// TIA Portal V17 export
// export: Created 2024-09-02T12:50:24.6153138Z, ExportSetting WithDefaults, DisplayName Totally Integrated Automation Portal, DisplayVersion V17, DisplayName TIA Portal Openness, DisplayVersion V17, DisplayName TIA Portal Version Control Interface, DisplayVersion V17, DisplayName STEP 7 Professional, DisplayVersion V17, DisplayName STEP 7 Safety, DisplayVersion V17, DisplayName WinCC Professional, DisplayVersion V17
FUNCTION "Energy_And_Air_Counter" : Void   // FC23, LAD
{ S7_Optimized_Access := 'TRUE' }
VERSION : 0.1
// stored: AutoNumber false, IsIECCheckEnabled false, SetENOAutomatically false, UDAEnableTagReadback false
   VAR_INPUT
      Active_Air : DInt;
      Active_Energy : LReal;
      Reset_total : Bool;
      Reset_Time_Stamp : Bool;
      Count_Part : Bool;
   END_VAR
   VAR_TEMP
      Active_En_KWh : LReal;
      Active_En_M3 : Real;
      tActive_En_M3 : Real;
      Reset_periods_Energy : Bool;
      Number : Int;
      temp : Int;
      t_Move_data : Bool;
      tReset_total : Bool;
   END_VAR
   VAR_TEMP   // added for the SCL form of the ladder/FBD networks
      _w1 : Bool;
      _w2 : Bool;
      _w3 : Bool;
   END_VAR
BEGIN

REGION Network 1: Actual_Active_Energy
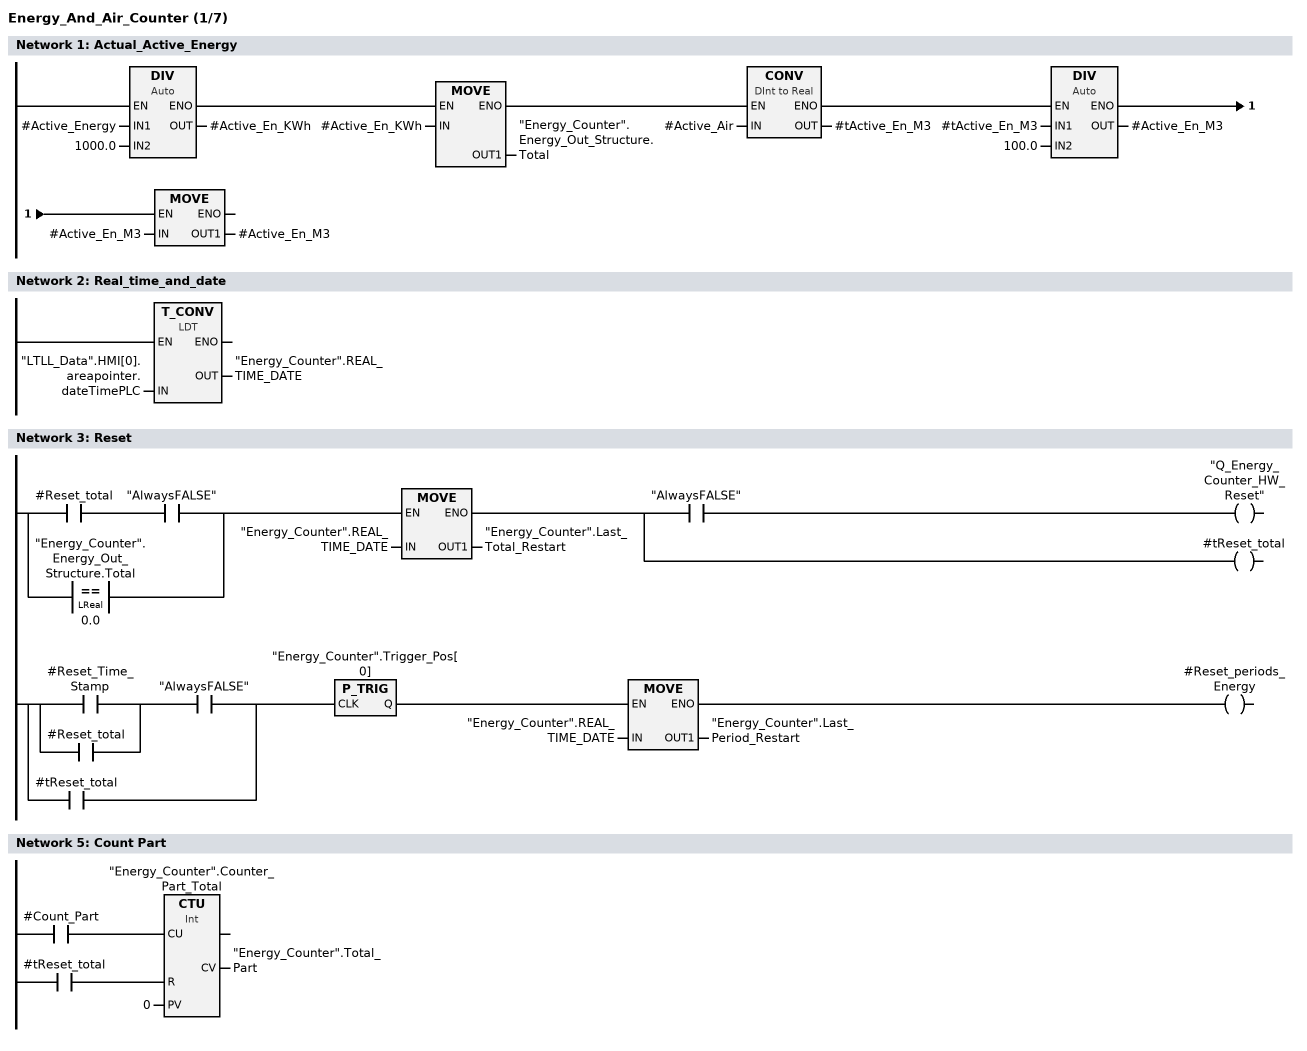
   RUNG wire#powerrail
      Div(in1 := #Active_Energy, in2 := 1000.0, out => #Active_En_KWh)
      Move(in := #Active_En_KWh, out1 => "Energy_Counter".Energy_Out_Structure.Total)
      { S7_Templates := "[SrcType := DInt, DestType := Real]" } Convert(in := #Active_Air, out => #tActive_En_M3)
      Div(in1 := #tActive_En_M3, in2 := 100.0, out => #Active_En_M3)
      Move(in := #Active_En_M3, out1 => #Active_En_M3)
   END_RUNG
   // the same network as SCL:
   #Active_En_KWh := #Active_Energy / 1000.0;
   "Energy_Counter".Energy_Out_Structure.Total := #Active_En_KWh;
   #tActive_En_M3 := DINT_TO_REAL(#Active_Air);
   #Active_En_M3 := #tActive_En_M3 / 100.0;
   #Active_En_M3 := #Active_En_M3;
END_REGION

REGION Network 2: Real_time_and_date
   RUNG wire#powerrail
      { S7_Templates := "[src_type := LDT, dest_type := DTL]" } T_CONV(IN := "LTLL_Data".HMI[0].areapointer.dateTimePLC, OUT => "Energy_Counter".REAL_TIME_DATE)
   END_RUNG
   // the same network as SCL:
   T_CONV(IN := "LTLL_Data".HMI[0].areapointer.dateTimePLC, OUT => "Energy_Counter".REAL_TIME_DATE);
END_REGION

REGION Network 3: Reset
   RUNG wire#powerrail
      Contact( #Reset_total )
      Contact( "AlwaysFALSE" )
      wire#w1
      Move(in := "Energy_Counter".REAL_TIME_DATE, out1 => "Energy_Counter".Last_Total_Restart)
      wire#w2
      Contact( "AlwaysFALSE" )
      Coil( "Q_Energy_Counter_HW_Reset" )
   END_RUNG
   RUNG wire#powerrail
      { S7_Templates := "SrcType := LReal" } EQ_Contact(in1 := "Energy_Counter".Energy_Out_Structure.Total, in2 := 0.0)
   END_RUNG wire#w1
   RUNG wire#w2
      Coil( #tReset_total )
   END_RUNG
   RUNG wire#powerrail
      Contact( #Reset_Time_Stamp )
      wire#w3
      Contact( "AlwaysFALSE" )
      wire#w4
      P_Trig( "Energy_Counter".Trigger_Pos[0] )
      Move(in := "Energy_Counter".REAL_TIME_DATE, out1 => "Energy_Counter".Last_Period_Restart)
      Coil( #Reset_periods_Energy )
   END_RUNG
   RUNG wire#powerrail
      Contact( #Reset_total )
   END_RUNG wire#w3
   RUNG wire#powerrail
      Contact( #tReset_total )
   END_RUNG wire#w4
   // the same network as SCL:
   #_w1 := (#Reset_total AND "AlwaysFALSE") OR ("Energy_Counter".Energy_Out_Structure.Total = 0.0);
   IF #_w1 THEN "Energy_Counter".Last_Total_Restart := "Energy_Counter".REAL_TIME_DATE; END_IF;
   "Q_Energy_Counter_HW_Reset" := #_w1 AND "AlwaysFALSE";
   #tReset_total := #_w1;
   #_w2 := ((#Reset_Time_Stamp OR #Reset_total) AND "AlwaysFALSE") OR #tReset_total;
   #_w3 := #_w2 AND NOT "Energy_Counter".Trigger_Pos[0];   // rising edge
   "Energy_Counter".Trigger_Pos[0] := #_w2;
   IF #_w3 THEN "Energy_Counter".Last_Period_Restart := "Energy_Counter".REAL_TIME_DATE; END_IF;
   #Reset_periods_Energy := #_w3;
END_REGION

REGION Network 4: ########### Part Counting #########
END_REGION

REGION Network 5: Count Part
   RUNG wire#powerrail
      Contact( #Count_Part )
      { S7_Templates := "value_type := Int" } "Energy_Counter".Counter_Part_Total.CTU(r := wire#w1, pv := 0, cv => "Energy_Counter".Total_Part)
   END_RUNG
   RUNG wire#powerrail
      Contact( #tReset_total )
   END_RUNG wire#w1
   // the same network as SCL:
   "Energy_Counter".Counter_Part_Total.CTU(CU := #Count_Part,
                           R := #tReset_total,
                           PV := 0,
                           CV => "Energy_Counter".Total_Part);
END_REGION

REGION Network 6: Total Energi / Air per Part
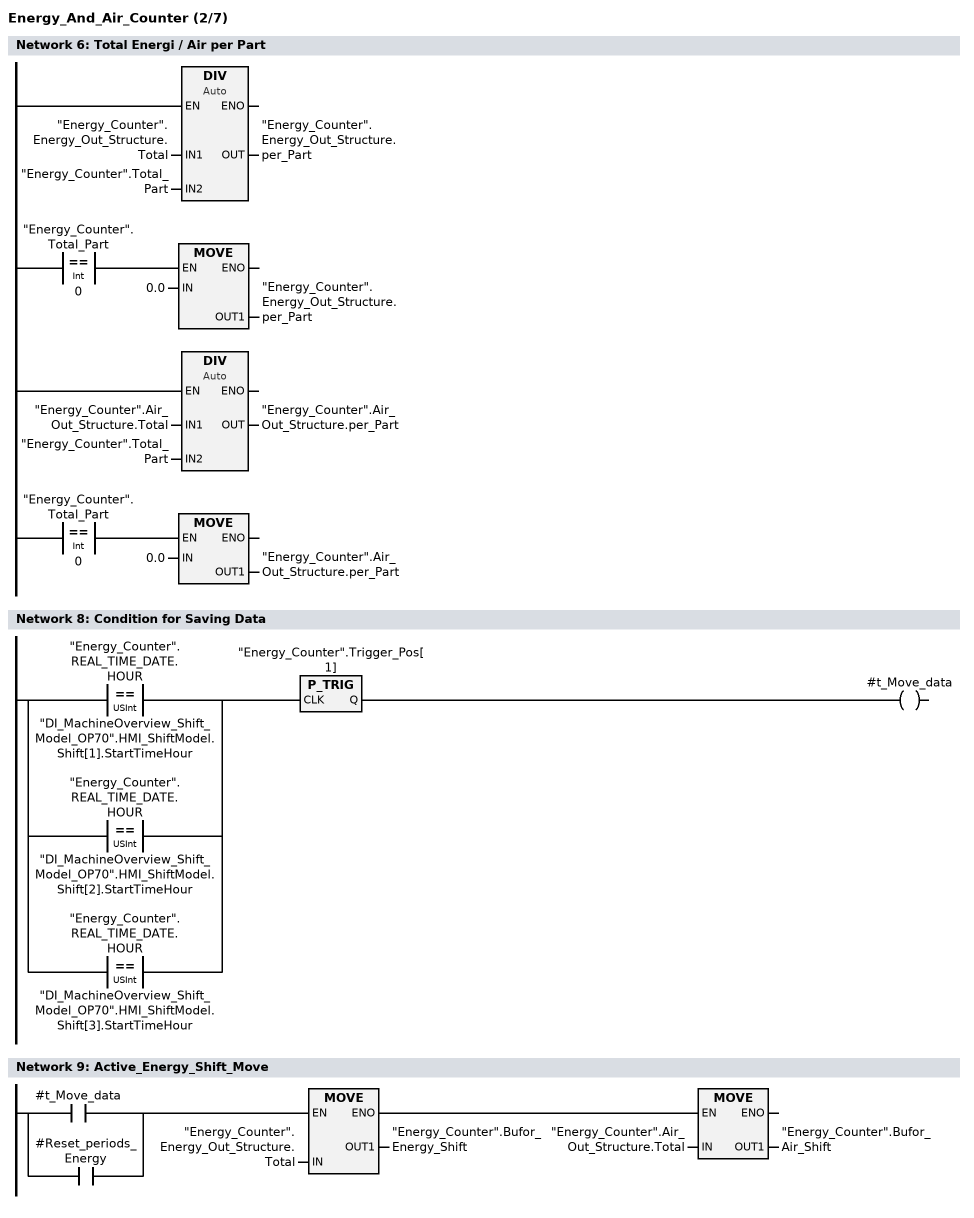
   RUNG wire#powerrail
      Div(in1 := "Energy_Counter".Energy_Out_Structure.Total, in2 := "Energy_Counter".Total_Part, out => "Energy_Counter".Energy_Out_Structure.per_Part)
   END_RUNG
   RUNG wire#powerrail
      { S7_Templates := "SrcType := Int" } EQ_Contact(in1 := "Energy_Counter".Total_Part, in2 := 0)
      Move(in := 0.0, out1 => "Energy_Counter".Energy_Out_Structure.per_Part)
   END_RUNG
   RUNG wire#powerrail
      Div(in1 := "Energy_Counter".Air_Out_Structure.Total, in2 := "Energy_Counter".Total_Part, out => "Energy_Counter".Air_Out_Structure.per_Part)
   END_RUNG
   RUNG wire#powerrail
      { S7_Templates := "SrcType := Int" } EQ_Contact(in1 := "Energy_Counter".Total_Part, in2 := 0)
      Move(in := 0.0, out1 => "Energy_Counter".Air_Out_Structure.per_Part)
   END_RUNG
   // the same network as SCL:
   "Energy_Counter".Energy_Out_Structure.per_Part := "Energy_Counter".Energy_Out_Structure.Total / "Energy_Counter".Total_Part;
   IF "Energy_Counter".Total_Part = 0 THEN "Energy_Counter".Energy_Out_Structure.per_Part := 0.0; END_IF;
   "Energy_Counter".Air_Out_Structure.per_Part := "Energy_Counter".Air_Out_Structure.Total / "Energy_Counter".Total_Part;
   IF "Energy_Counter".Total_Part = 0 THEN "Energy_Counter".Air_Out_Structure.per_Part := 0.0; END_IF;
END_REGION

REGION Network 7: ########### ENERGY PER SHIFT #########
END_REGION

REGION Network 8: Condition for Saving Data
   RUNG wire#powerrail
      { S7_Templates := "SrcType := USInt" } EQ_Contact(in1 := "Energy_Counter".REAL_TIME_DATE.HOUR, in2 := "DI_MachineOverview_Shift_Model_OP70".HMI_ShiftModel.Shift[1].StartTimeHour)
      wire#w1
      P_Trig( "Energy_Counter".Trigger_Pos[1] )
      Coil( #t_Move_data )
   END_RUNG
   RUNG wire#powerrail
      { S7_Templates := "SrcType := USInt" } EQ_Contact(in1 := "Energy_Counter".REAL_TIME_DATE.HOUR, in2 := "DI_MachineOverview_Shift_Model_OP70".HMI_ShiftModel.Shift[2].StartTimeHour)
   END_RUNG wire#w1
   RUNG wire#powerrail
      { S7_Templates := "SrcType := USInt" } EQ_Contact(in1 := "Energy_Counter".REAL_TIME_DATE.HOUR, in2 := "DI_MachineOverview_Shift_Model_OP70".HMI_ShiftModel.Shift[3].StartTimeHour)
   END_RUNG wire#w1
   // the same network as SCL:
   #_w1 := ("Energy_Counter".REAL_TIME_DATE.HOUR = "DI_MachineOverview_Shift_Model_OP70".HMI_ShiftModel.Shift[1].StartTimeHour) OR ("Energy_Counter".REAL_TIME_DATE.HOUR = "DI_MachineOverview_Shift_Model_OP70".HMI_ShiftModel.Shift[2].StartTimeHour) OR ("Energy_Counter".REAL_TIME_DATE.HOUR = "DI_MachineOverview_Shift_Model_OP70".HMI_ShiftModel.Shift[3].StartTimeHour);
   #_w2 := #_w1 AND NOT "Energy_Counter".Trigger_Pos[1];   // rising edge
   "Energy_Counter".Trigger_Pos[1] := #_w1;
   #t_Move_data := #_w2;
END_REGION

REGION Network 9: Active_Energy_Shift_Move
   RUNG wire#powerrail
      Contact( #t_Move_data )
      wire#w1
      Move(in := "Energy_Counter".Energy_Out_Structure.Total, out1 => "Energy_Counter".Bufor_Energy_Shift)
      Move(in := "Energy_Counter".Air_Out_Structure.Total, out1 => "Energy_Counter".Bufor_Air_Shift)
   END_RUNG
   RUNG wire#powerrail
      Contact( #Reset_periods_Energy )
   END_RUNG wire#w1
   // the same network as SCL:
   IF #t_Move_data OR #Reset_periods_Energy THEN
       "Energy_Counter".Bufor_Energy_Shift := "Energy_Counter".Energy_Out_Structure.Total;
       "Energy_Counter".Bufor_Air_Shift := "Energy_Counter".Air_Out_Structure.Total;
   END_IF;
END_REGION

REGION Network 10: Calculation
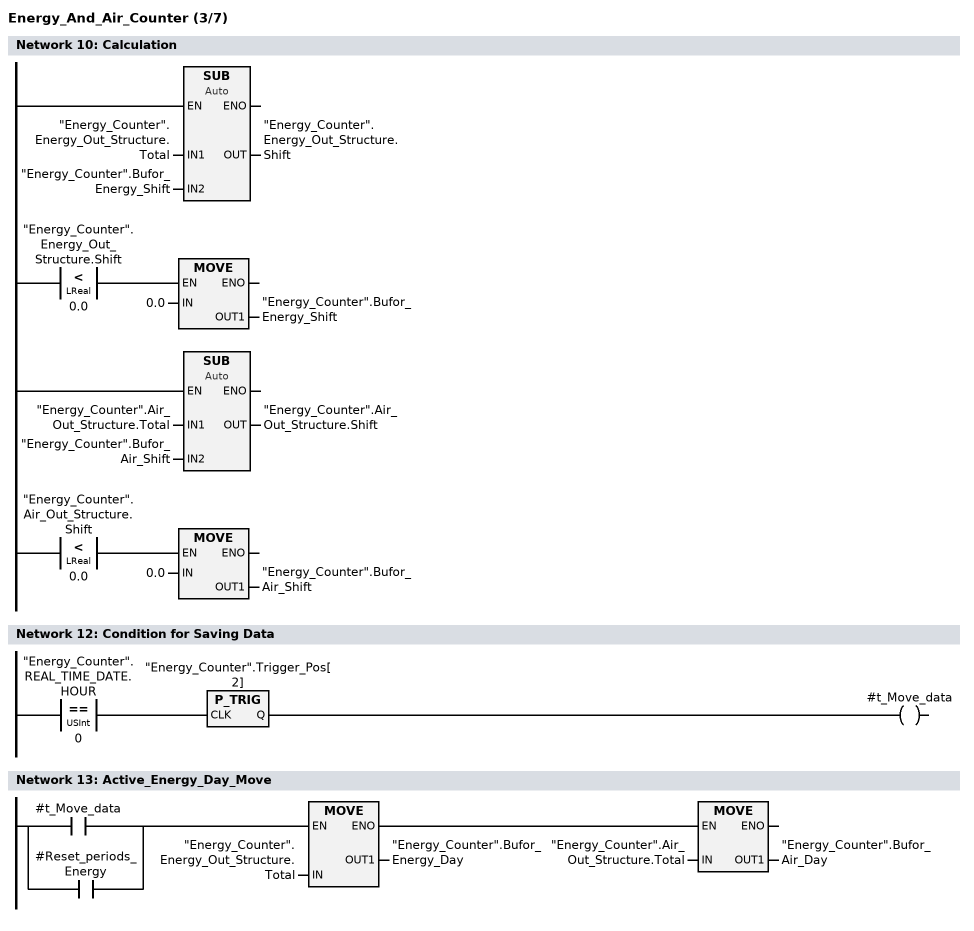
   RUNG wire#powerrail
      Sub(in1 := "Energy_Counter".Energy_Out_Structure.Total, in2 := "Energy_Counter".Bufor_Energy_Shift, out => "Energy_Counter".Energy_Out_Structure.Shift)
   END_RUNG
   RUNG wire#powerrail
      { S7_Templates := "SrcType := LReal" } LT_Contact(in1 := "Energy_Counter".Energy_Out_Structure.Shift, in2 := 0.0)
      Move(in := 0.0, out1 => "Energy_Counter".Bufor_Energy_Shift)
   END_RUNG
   RUNG wire#powerrail
      Sub(in1 := "Energy_Counter".Air_Out_Structure.Total, in2 := "Energy_Counter".Bufor_Air_Shift, out => "Energy_Counter".Air_Out_Structure.Shift)
   END_RUNG
   RUNG wire#powerrail
      { S7_Templates := "SrcType := LReal" } LT_Contact(in1 := "Energy_Counter".Air_Out_Structure.Shift, in2 := 0.0)
      Move(in := 0.0, out1 => "Energy_Counter".Bufor_Air_Shift)
   END_RUNG
   // the same network as SCL:
   "Energy_Counter".Energy_Out_Structure.Shift := "Energy_Counter".Energy_Out_Structure.Total - "Energy_Counter".Bufor_Energy_Shift;
   IF "Energy_Counter".Energy_Out_Structure.Shift < 0.0 THEN
       "Energy_Counter".Bufor_Energy_Shift := 0.0;
   END_IF;
   "Energy_Counter".Air_Out_Structure.Shift := "Energy_Counter".Air_Out_Structure.Total - "Energy_Counter".Bufor_Air_Shift;
   IF "Energy_Counter".Air_Out_Structure.Shift < 0.0 THEN "Energy_Counter".Bufor_Air_Shift := 0.0; END_IF;
END_REGION

REGION Network 11: ########### ENERGY PER DAY #########
END_REGION

REGION Network 12: Condition for Saving Data
   RUNG wire#powerrail
      { S7_Templates := "SrcType := USInt" } EQ_Contact(in1 := "Energy_Counter".REAL_TIME_DATE.HOUR, in2 := 0)
      P_Trig( "Energy_Counter".Trigger_Pos[2] )
      Coil( #t_Move_data )
   END_RUNG
   // the same network as SCL:
   #_w1 := "Energy_Counter".REAL_TIME_DATE.HOUR = 0;
   #_w2 := #_w1 AND NOT "Energy_Counter".Trigger_Pos[2];   // rising edge
   "Energy_Counter".Trigger_Pos[2] := #_w1;
   #t_Move_data := #_w2;
END_REGION

REGION Network 13: Active_Energy_Day_Move
   RUNG wire#powerrail
      Contact( #t_Move_data )
      wire#w1
      Move(in := "Energy_Counter".Energy_Out_Structure.Total, out1 => "Energy_Counter".Bufor_Energy_Day)
      Move(in := "Energy_Counter".Air_Out_Structure.Total, out1 => "Energy_Counter".Bufor_Air_Day)
   END_RUNG
   RUNG wire#powerrail
      Contact( #Reset_periods_Energy )
   END_RUNG wire#w1
   // the same network as SCL:
   IF #t_Move_data OR #Reset_periods_Energy THEN
       "Energy_Counter".Bufor_Energy_Day := "Energy_Counter".Energy_Out_Structure.Total;
       "Energy_Counter".Bufor_Air_Day := "Energy_Counter".Air_Out_Structure.Total;
   END_IF;
END_REGION

REGION Network 14: Calculation
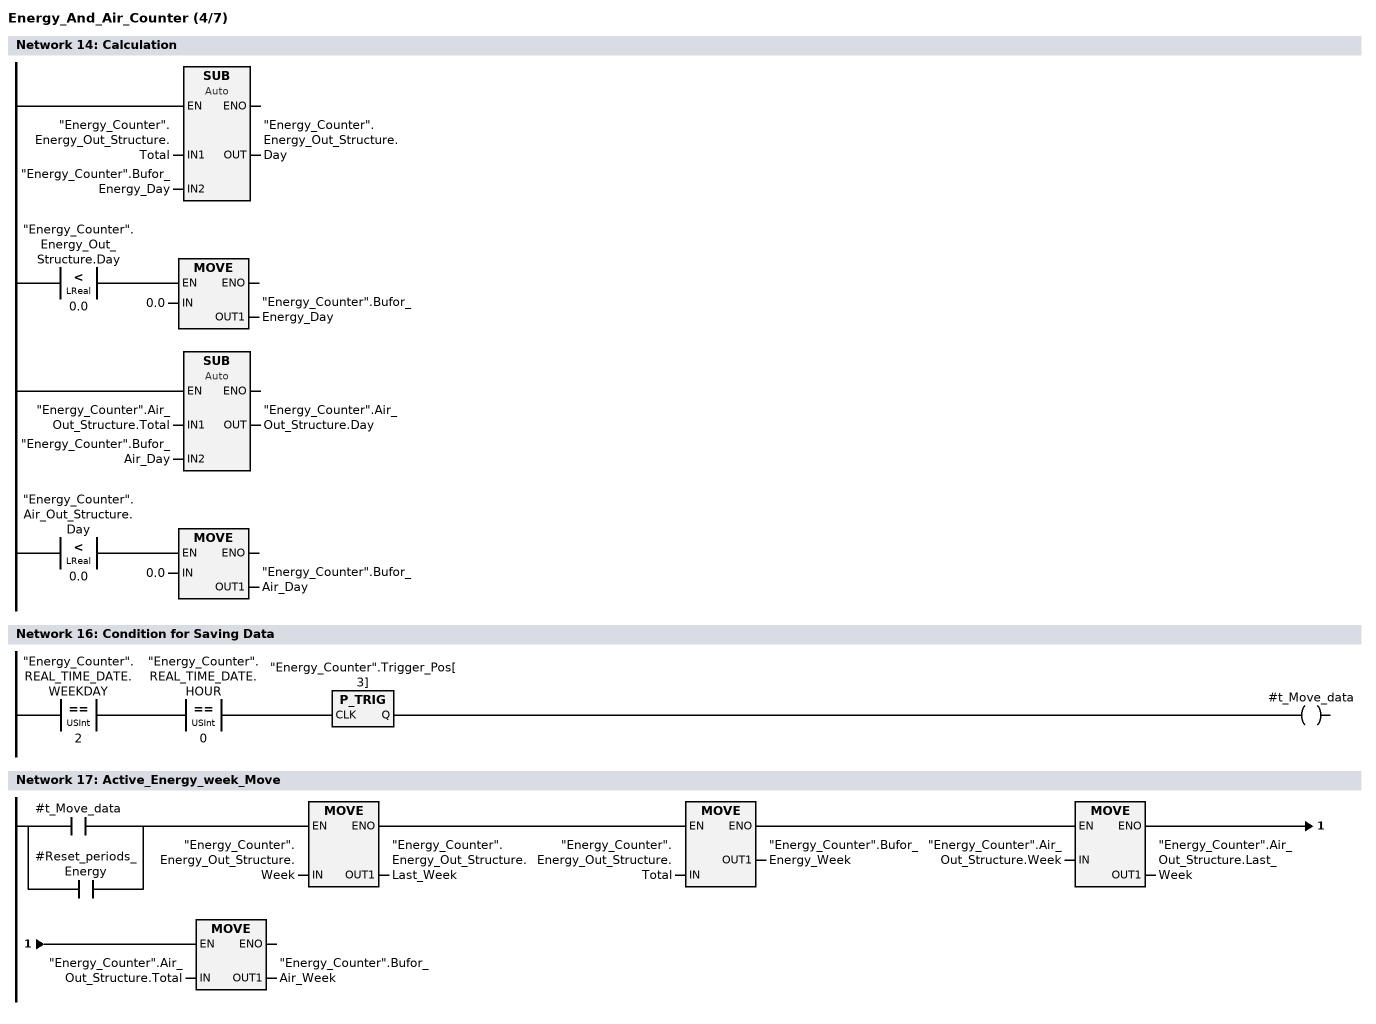
   RUNG wire#powerrail
      Sub(in1 := "Energy_Counter".Energy_Out_Structure.Total, in2 := "Energy_Counter".Bufor_Energy_Day, out => "Energy_Counter".Energy_Out_Structure.Day)
   END_RUNG
   RUNG wire#powerrail
      { S7_Templates := "SrcType := LReal" } LT_Contact(in1 := "Energy_Counter".Energy_Out_Structure.Day, in2 := 0.0)
      Move(in := 0.0, out1 => "Energy_Counter".Bufor_Energy_Day)
   END_RUNG
   RUNG wire#powerrail
      Sub(in1 := "Energy_Counter".Air_Out_Structure.Total, in2 := "Energy_Counter".Bufor_Air_Day, out => "Energy_Counter".Air_Out_Structure.Day)
   END_RUNG
   RUNG wire#powerrail
      { S7_Templates := "SrcType := LReal" } LT_Contact(in1 := "Energy_Counter".Air_Out_Structure.Day, in2 := 0.0)
      Move(in := 0.0, out1 => "Energy_Counter".Bufor_Air_Day)
   END_RUNG
   // the same network as SCL:
   "Energy_Counter".Energy_Out_Structure.Day := "Energy_Counter".Energy_Out_Structure.Total - "Energy_Counter".Bufor_Energy_Day;
   IF "Energy_Counter".Energy_Out_Structure.Day < 0.0 THEN "Energy_Counter".Bufor_Energy_Day := 0.0; END_IF;
   "Energy_Counter".Air_Out_Structure.Day := "Energy_Counter".Air_Out_Structure.Total - "Energy_Counter".Bufor_Air_Day;
   IF "Energy_Counter".Air_Out_Structure.Day < 0.0 THEN "Energy_Counter".Bufor_Air_Day := 0.0; END_IF;
END_REGION

REGION Network 15: ########### ENERGY PER WEEK #########
END_REGION

REGION Network 16: Condition for Saving Data
   RUNG wire#powerrail
      { S7_Templates := "SrcType := USInt" } EQ_Contact(in1 := "Energy_Counter".REAL_TIME_DATE.WEEKDAY, in2 := 2)
      { S7_Templates := "SrcType := USInt" } EQ_Contact(in1 := "Energy_Counter".REAL_TIME_DATE.HOUR, in2 := 0)
      P_Trig( "Energy_Counter".Trigger_Pos[3] )
      Coil( #t_Move_data )
   END_RUNG
   // the same network as SCL:
   #_w1 := ("Energy_Counter".REAL_TIME_DATE.WEEKDAY = 2) AND ("Energy_Counter".REAL_TIME_DATE.HOUR = 0);
   #_w2 := #_w1 AND NOT "Energy_Counter".Trigger_Pos[3];   // rising edge
   "Energy_Counter".Trigger_Pos[3] := #_w1;
   #t_Move_data := #_w2;
END_REGION

REGION Network 17: Active_Energy_week_Move
   RUNG wire#powerrail
      Contact( #t_Move_data )
      wire#w1
      Move(in := "Energy_Counter".Energy_Out_Structure.Week, out1 => "Energy_Counter".Energy_Out_Structure.Last_Week)
      Move(in := "Energy_Counter".Energy_Out_Structure.Total, out1 => "Energy_Counter".Bufor_Energy_Week)
      Move(in := "Energy_Counter".Air_Out_Structure.Week, out1 => "Energy_Counter".Air_Out_Structure.Last_Week)
      Move(in := "Energy_Counter".Air_Out_Structure.Total, out1 => "Energy_Counter".Bufor_Air_Week)
   END_RUNG
   RUNG wire#powerrail
      Contact( #Reset_periods_Energy )
   END_RUNG wire#w1
   // the same network as SCL:
   IF #t_Move_data OR #Reset_periods_Energy THEN
       "Energy_Counter".Energy_Out_Structure.Last_Week := "Energy_Counter".Energy_Out_Structure.Week;
       "Energy_Counter".Bufor_Energy_Week := "Energy_Counter".Energy_Out_Structure.Total;
       "Energy_Counter".Air_Out_Structure.Last_Week := "Energy_Counter".Air_Out_Structure.Week;
       "Energy_Counter".Bufor_Air_Week := "Energy_Counter".Air_Out_Structure.Total;
   END_IF;
END_REGION

REGION Network 18: Calculation
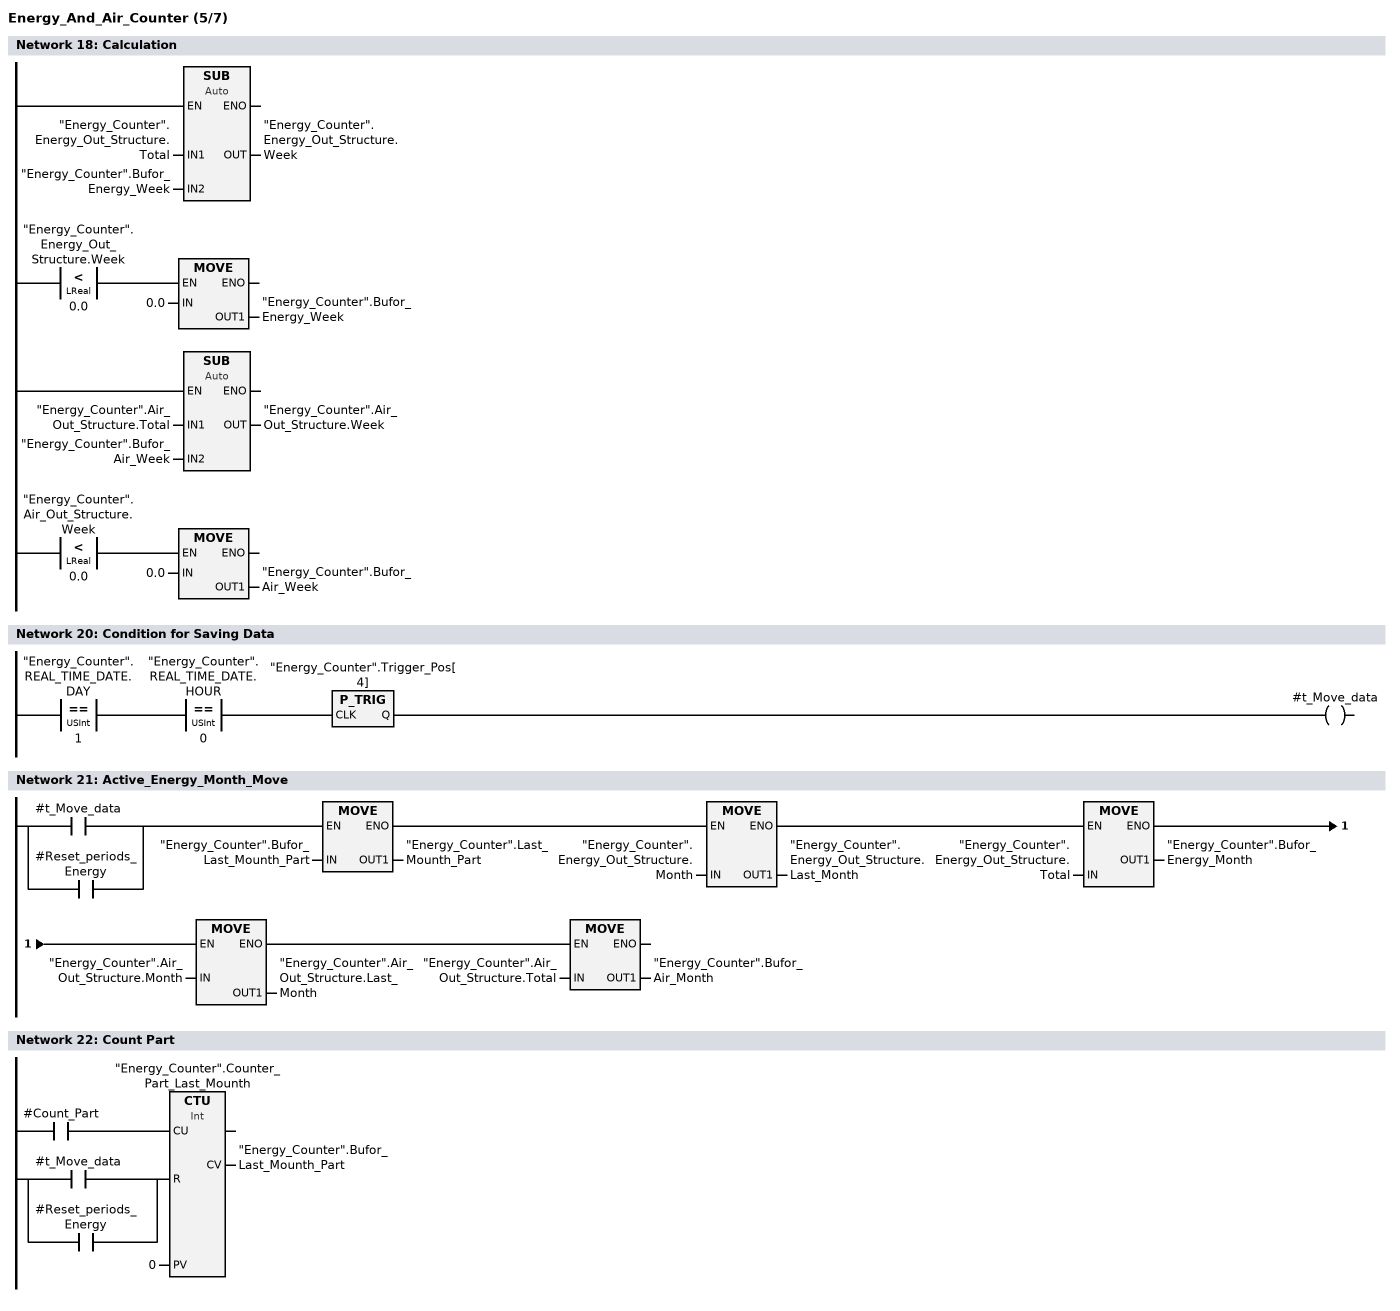
   RUNG wire#powerrail
      Sub(in1 := "Energy_Counter".Energy_Out_Structure.Total, in2 := "Energy_Counter".Bufor_Energy_Week, out => "Energy_Counter".Energy_Out_Structure.Week)
   END_RUNG
   RUNG wire#powerrail
      { S7_Templates := "SrcType := LReal" } LT_Contact(in1 := "Energy_Counter".Energy_Out_Structure.Week, in2 := 0.0)
      Move(in := 0.0, out1 => "Energy_Counter".Bufor_Energy_Week)
   END_RUNG
   RUNG wire#powerrail
      Sub(in1 := "Energy_Counter".Air_Out_Structure.Total, in2 := "Energy_Counter".Bufor_Air_Week, out => "Energy_Counter".Air_Out_Structure.Week)
   END_RUNG
   RUNG wire#powerrail
      { S7_Templates := "SrcType := LReal" } LT_Contact(in1 := "Energy_Counter".Air_Out_Structure.Week, in2 := 0.0)
      Move(in := 0.0, out1 => "Energy_Counter".Bufor_Air_Week)
   END_RUNG
   // the same network as SCL:
   "Energy_Counter".Energy_Out_Structure.Week := "Energy_Counter".Energy_Out_Structure.Total - "Energy_Counter".Bufor_Energy_Week;
   IF "Energy_Counter".Energy_Out_Structure.Week < 0.0 THEN
       "Energy_Counter".Bufor_Energy_Week := 0.0;
   END_IF;
   "Energy_Counter".Air_Out_Structure.Week := "Energy_Counter".Air_Out_Structure.Total - "Energy_Counter".Bufor_Air_Week;
   IF "Energy_Counter".Air_Out_Structure.Week < 0.0 THEN "Energy_Counter".Bufor_Air_Week := 0.0; END_IF;
END_REGION

REGION Network 19: ########### ENERGY PER MONTH #########
END_REGION

REGION Network 20: Condition for Saving Data
   RUNG wire#powerrail
      { S7_Templates := "SrcType := USInt" } EQ_Contact(in1 := "Energy_Counter".REAL_TIME_DATE.DAY, in2 := 1)
      { S7_Templates := "SrcType := USInt" } EQ_Contact(in1 := "Energy_Counter".REAL_TIME_DATE.HOUR, in2 := 0)
      P_Trig( "Energy_Counter".Trigger_Pos[4] )
      Coil( #t_Move_data )
   END_RUNG
   // the same network as SCL:
   #_w1 := ("Energy_Counter".REAL_TIME_DATE.DAY = 1) AND ("Energy_Counter".REAL_TIME_DATE.HOUR = 0);
   #_w2 := #_w1 AND NOT "Energy_Counter".Trigger_Pos[4];   // rising edge
   "Energy_Counter".Trigger_Pos[4] := #_w1;
   #t_Move_data := #_w2;
END_REGION

REGION Network 21: Active_Energy_Month_Move
   RUNG wire#powerrail
      Contact( #t_Move_data )
      wire#w1
      Move(in := "Energy_Counter".Bufor_Last_Mounth_Part, out1 => "Energy_Counter".Last_Mounth_Part)
      Move(in := "Energy_Counter".Energy_Out_Structure.Month, out1 => "Energy_Counter".Energy_Out_Structure.Last_Month)
      Move(in := "Energy_Counter".Energy_Out_Structure.Total, out1 => "Energy_Counter".Bufor_Energy_Month)
      Move(in := "Energy_Counter".Air_Out_Structure.Month, out1 => "Energy_Counter".Air_Out_Structure.Last_Month)
      Move(in := "Energy_Counter".Air_Out_Structure.Total, out1 => "Energy_Counter".Bufor_Air_Month)
   END_RUNG
   RUNG wire#powerrail
      Contact( #Reset_periods_Energy )
   END_RUNG wire#w1
   // the same network as SCL:
   IF #t_Move_data OR #Reset_periods_Energy THEN
       "Energy_Counter".Last_Mounth_Part := "Energy_Counter".Bufor_Last_Mounth_Part;
       "Energy_Counter".Energy_Out_Structure.Last_Month := "Energy_Counter".Energy_Out_Structure.Month;
       "Energy_Counter".Bufor_Energy_Month := "Energy_Counter".Energy_Out_Structure.Total;
       "Energy_Counter".Air_Out_Structure.Last_Month := "Energy_Counter".Air_Out_Structure.Month;
       "Energy_Counter".Bufor_Air_Month := "Energy_Counter".Air_Out_Structure.Total;
   END_IF;
END_REGION

REGION Network 22: Count Part
   RUNG wire#powerrail
      Contact( #Count_Part )
      { S7_Templates := "value_type := Int" } "Energy_Counter".Counter_Part_Last_Mounth.CTU(r := wire#w1, pv := 0, cv => "Energy_Counter".Bufor_Last_Mounth_Part)
   END_RUNG
   RUNG wire#powerrail
      Contact( #t_Move_data )
   END_RUNG wire#w1
   RUNG wire#powerrail
      Contact( #Reset_periods_Energy )
   END_RUNG wire#w1
   // the same network as SCL:
   "Energy_Counter".Counter_Part_Last_Mounth.CTU(CU := #Count_Part,
                           R := #t_Move_data OR #Reset_periods_Energy,
                           PV := 0,
                           CV => "Energy_Counter".Bufor_Last_Mounth_Part);
END_REGION

REGION Network 23: Calculation
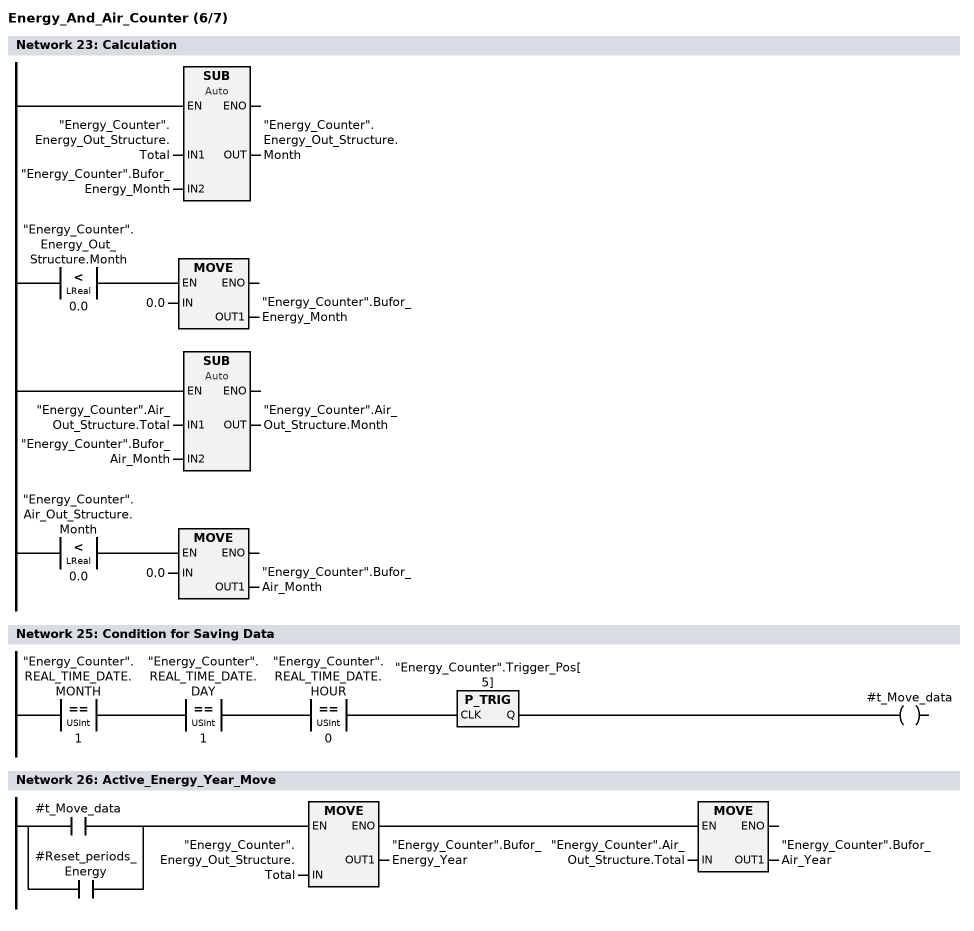
   RUNG wire#powerrail
      Sub(in1 := "Energy_Counter".Energy_Out_Structure.Total, in2 := "Energy_Counter".Bufor_Energy_Month, out => "Energy_Counter".Energy_Out_Structure.Month)
   END_RUNG
   RUNG wire#powerrail
      { S7_Templates := "SrcType := LReal" } LT_Contact(in1 := "Energy_Counter".Energy_Out_Structure.Month, in2 := 0.0)
      Move(in := 0.0, out1 => "Energy_Counter".Bufor_Energy_Month)
   END_RUNG
   RUNG wire#powerrail
      Sub(in1 := "Energy_Counter".Air_Out_Structure.Total, in2 := "Energy_Counter".Bufor_Air_Month, out => "Energy_Counter".Air_Out_Structure.Month)
   END_RUNG
   RUNG wire#powerrail
      { S7_Templates := "SrcType := LReal" } LT_Contact(in1 := "Energy_Counter".Air_Out_Structure.Month, in2 := 0.0)
      Move(in := 0.0, out1 => "Energy_Counter".Bufor_Air_Month)
   END_RUNG
   // the same network as SCL:
   "Energy_Counter".Energy_Out_Structure.Month := "Energy_Counter".Energy_Out_Structure.Total - "Energy_Counter".Bufor_Energy_Month;
   IF "Energy_Counter".Energy_Out_Structure.Month < 0.0 THEN
       "Energy_Counter".Bufor_Energy_Month := 0.0;
   END_IF;
   "Energy_Counter".Air_Out_Structure.Month := "Energy_Counter".Air_Out_Structure.Total - "Energy_Counter".Bufor_Air_Month;
   IF "Energy_Counter".Air_Out_Structure.Month < 0.0 THEN "Energy_Counter".Bufor_Air_Month := 0.0; END_IF;
END_REGION

REGION Network 24: ########### ENERGY PER YEAR#########
END_REGION

REGION Network 25: Condition for Saving Data
   RUNG wire#powerrail
      { S7_Templates := "SrcType := USInt" } EQ_Contact(in1 := "Energy_Counter".REAL_TIME_DATE.MONTH, in2 := 1)
      { S7_Templates := "SrcType := USInt" } EQ_Contact(in1 := "Energy_Counter".REAL_TIME_DATE.DAY, in2 := 1)
      { S7_Templates := "SrcType := USInt" } EQ_Contact(in1 := "Energy_Counter".REAL_TIME_DATE.HOUR, in2 := 0)
      P_Trig( "Energy_Counter".Trigger_Pos[5] )
      Coil( #t_Move_data )
   END_RUNG
   // the same network as SCL:
   #_w1 := ("Energy_Counter".REAL_TIME_DATE.MONTH = 1) AND ("Energy_Counter".REAL_TIME_DATE.DAY = 1) AND ("Energy_Counter".REAL_TIME_DATE.HOUR = 0);
   #_w2 := #_w1 AND NOT "Energy_Counter".Trigger_Pos[5];   // rising edge
   "Energy_Counter".Trigger_Pos[5] := #_w1;
   #t_Move_data := #_w2;
END_REGION

REGION Network 26: Active_Energy_Year_Move
   RUNG wire#powerrail
      Contact( #t_Move_data )
      wire#w1
      Move(in := "Energy_Counter".Energy_Out_Structure.Total, out1 => "Energy_Counter".Bufor_Energy_Year)
      Move(in := "Energy_Counter".Air_Out_Structure.Total, out1 => "Energy_Counter".Bufor_Air_Year)
   END_RUNG
   RUNG wire#powerrail
      Contact( #Reset_periods_Energy )
   END_RUNG wire#w1
   // the same network as SCL:
   IF #t_Move_data OR #Reset_periods_Energy THEN
       "Energy_Counter".Bufor_Energy_Year := "Energy_Counter".Energy_Out_Structure.Total;
       "Energy_Counter".Bufor_Air_Year := "Energy_Counter".Air_Out_Structure.Total;
   END_IF;
END_REGION

REGION Network 27: Calculation
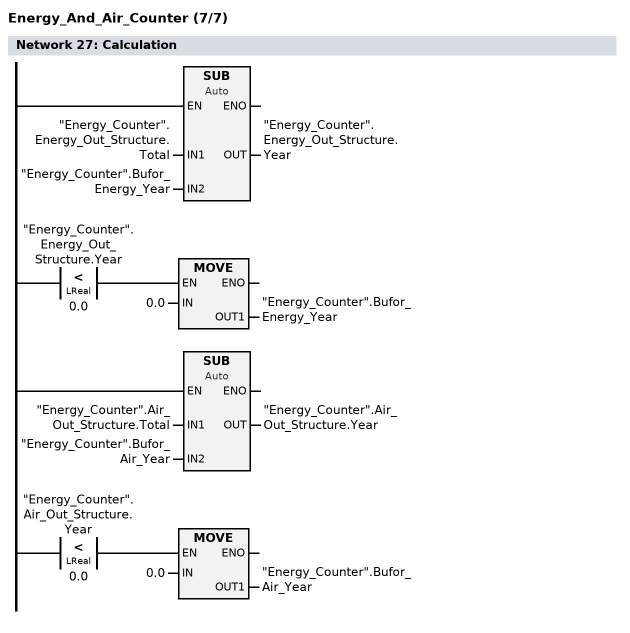
   RUNG wire#powerrail
      Sub(in1 := "Energy_Counter".Energy_Out_Structure.Total, in2 := "Energy_Counter".Bufor_Energy_Year, out => "Energy_Counter".Energy_Out_Structure.Year)
   END_RUNG
   RUNG wire#powerrail
      { S7_Templates := "SrcType := LReal" } LT_Contact(in1 := "Energy_Counter".Energy_Out_Structure.Year, in2 := 0.0)
      Move(in := 0.0, out1 => "Energy_Counter".Bufor_Energy_Year)
   END_RUNG
   RUNG wire#powerrail
      Sub(in1 := "Energy_Counter".Air_Out_Structure.Total, in2 := "Energy_Counter".Bufor_Air_Year, out => "Energy_Counter".Air_Out_Structure.Year)
   END_RUNG
   RUNG wire#powerrail
      { S7_Templates := "SrcType := LReal" } LT_Contact(in1 := "Energy_Counter".Air_Out_Structure.Year, in2 := 0.0)
      Move(in := 0.0, out1 => "Energy_Counter".Bufor_Air_Year)
   END_RUNG
   // the same network as SCL:
   "Energy_Counter".Energy_Out_Structure.Year := "Energy_Counter".Energy_Out_Structure.Total - "Energy_Counter".Bufor_Energy_Year;
   IF "Energy_Counter".Energy_Out_Structure.Year < 0.0 THEN
       "Energy_Counter".Bufor_Energy_Year := 0.0;
   END_IF;
   "Energy_Counter".Air_Out_Structure.Year := "Energy_Counter".Air_Out_Structure.Total - "Energy_Counter".Bufor_Air_Year;
   IF "Energy_Counter".Air_Out_Structure.Year < 0.0 THEN "Energy_Counter".Bufor_Air_Year := 0.0; END_IF;
END_REGION
END_FUNCTION
